{attribute addProperty BoxType "CPXXXX-BK7902-0016"}
{attribute addProperty Id "Term_382_KL1002KL1002_D229A9CA00"}
{attribute addProperty CRC "2996104891"}
{attribute addProperty SizeInBites "0"}
{attribute addProperty SizeInBytes "0"}
TYPE A_0009_CPXXXX_BK1150_0016_B294EEBB EXTENDS CPXXXX_4487A81F :
STRUCT
	{attribute addProperty Name "Term_382_KL1002"}
	Term_382_KL1002 : KL1002_D229A9CA;
END_STRUCT
END_TYPE

(* stored: Version 1.2.0.0, ProductVersion 3.1.4024.9
   DUT A_0009_CPXXXX_BK1150_0016_B294EEBB: Id {112d3630-6337-4209-88e6-8007756bc405} *)
